// TIA Portal V17 export
// export: Created 2025-11-04T09:12:31.4471126Z, ExportSetting WithDefaults, DisplayName Totally Integrated Automation Portal, DisplayVersion V17 Update 6
VAR_GLOBAL   // PLC tag table "Station10_IO"
   EStop_OK AT %I0.0 : Bool;   // Emergency stop circuit healthy (NC) / Not-Halt-Kreis i.O. (Öffner)
   Pump1_Fbk AT %I0.1 : Bool;   // Coolant pump running feedback
   Pump1_Trip AT %I0.2 : Bool;
   Pump1_Run AT %Q0.0 : Bool;
   Y1_Open AT %Q0.1 : Bool;
   Y1_Opened AT %I0.3 : Bool;
   PT101 AT %IW64 : Int;   // Coolant pressure 0-10 bar
   AutoMode AT %M10.0 : Bool;
END_VAR
